PROGRAM Blink
VAR
	hvacBlink 	: FB_HVACBlink();
	bEnable		: BOOL;
	tTimeOn		: TIME := T#2S;
	tTimeOff 	: TIME := T#1S;
END_VAR

VAR_OUTPUT
	bBlink			: BOOL;
	tNextSwitching  :TIME;
END_VAR

hvacBlink(bEnable:=bEnable,
tTimeOn:=tTimeOn,
tTimeOff:=tTimeOff,
bBlink=>,
tNextSwitching=>);

END_PROGRAM

(* stored: Version 1.1.0.1, ProductVersion 3.1.4024.12
   POU Blink: Id {616ae6ef-83ff-46d5-a9d4-a976618ae8ef}, SpecialFunc None *)
